// TIA Portal V20 export
DATA_BLOCK "DB_S300SetPoint"   // DB21
// stored: MemoryReserve 100, Namespace Global
   VAR
      Line : Struct
         ProductionLine : Struct
            DirChange : Struct
               Conveyor : Array[_.gminProductionLine.._.gmaxProductionLine] of "Global.S300ForceMode";
            END_STRUCT;
         END_STRUCT;
      END_STRUCT;
   END_VAR
BEGIN
END_DATA_BLOCK
